Fanuc KAREL source: kd00008.KL

-- PROVISIONAL review KL for V1013-1; original PC SHA256 5d4ec54b5ac0a284899580b1895b8d3a7a6c838ebf27fa4c2dde5672317b0baa
-- Incomplete behavior may be omitted. Consult companion uncertainty JSON. Do not deploy.
PROGRAM KD00008
%NOLOCKGROUP
VAR
  I : INTEGER
  J : INTEGER
  B : BOOLEAN
  R : REAL
  S : STRING[80]
BEGIN
  -- UNRESOLVED_PC offsets 5-12; opcodes 9D,23
  -- UNRESOLVED_PC offsets 17-21; opcodes 7F
END KD00008
